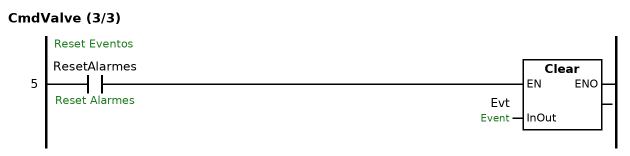
(* [picture p168: CmdValve, rungs 5-5] *)
(* Rung 5: Reset Eventos *)
IF ResetAlarmes THEN Clear(InOut := Evt); END_IF;
END_FUNCTION_BLOCK

FUNCTION_BLOCK CheckAlarmeEquip
VAR_IN_OUT
    Alm : Alarme;  (* Alarme *)
END_VAR
VAR_OUTPUT
    AlmOut : BOOL;  (* Output Alarme Agrupado *)
END_VAR
VAR_INPUT
    Enable : BOOL;
END_VAR
VAR_EXTERNAL
    ResetAlarmes : BOOL;
END_VAR
(* ladder, written here as Structured Text *)

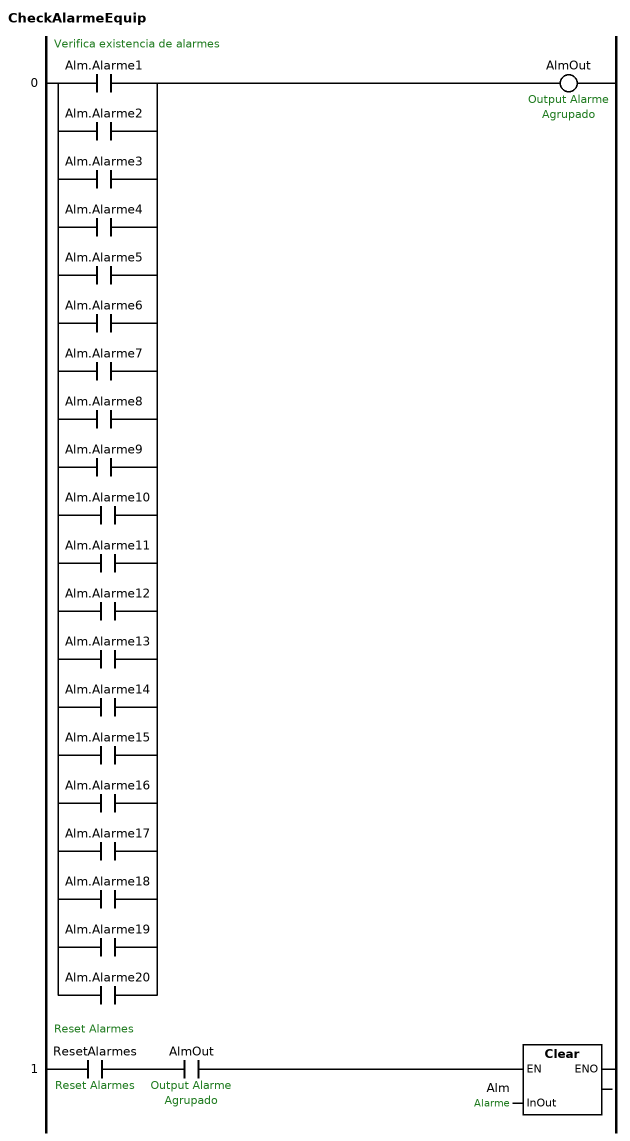
(* Rung 0: Verifica existencia de alarmes *)
AlmOut := Alm.Alarme1 OR Alm.Alarme2 OR Alm.Alarme3 OR Alm.Alarme4 OR Alm.Alarme5 OR Alm.Alarme6 OR Alm.Alarme7 OR Alm.Alarme8 OR Alm.Alarme9 OR Alm.Alarme10 OR Alm.Alarme11 OR Alm.Alarme12 OR Alm.Alarme13 OR Alm.Alarme14 OR Alm.Alarme15 OR Alm.Alarme16 OR Alm.Alarme17 OR Alm.Alarme18 OR Alm.Alarme19 OR Alm.Alarme20;
(* Rung 1: Reset Alarmes *)
IF ResetAlarmes AND AlmOut THEN Clear(InOut := Alm); END_IF;
END_FUNCTION_BLOCK

FUNCTION_BLOCK TimerPulse
VAR
    AuxTimeCalc : UINT;
END_VAR
VAR_INPUT
    Enable : BOOL;
    Pulse : BOOL;
    SetpointTime : UINT;
END_VAR
VAR
    _e1 : R_TRIG;
END_VAR
(* ladder, written here as Structured Text *)

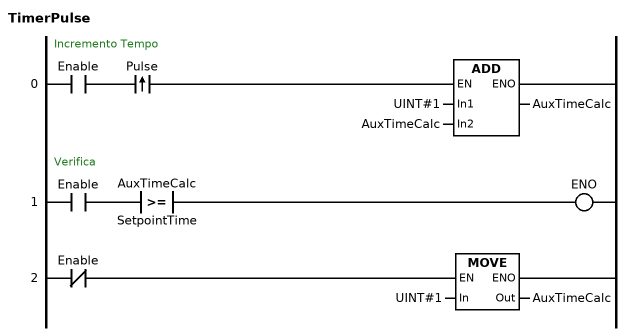
(* Rung 0: Incremento Tempo *)
_e1(CLK := Pulse);
IF Enable AND _e1.Q THEN AuxTimeCalc := UINT#1 + AuxTimeCalc; END_IF;
(* Rung 1: Verifica *)
ENO := Enable AND (AuxTimeCalc >= SetpointTime);
(* Rung 2 *)
IF NOT Enable THEN AuxTimeCalc := UINT#1; END_IF;
END_FUNCTION_BLOCK

FUNCTION_BLOCK EAN13Read
VAR
    SomaPares : UINT;
    SomaImpares : UINT;
    Resto : UINT;
    G_Step05 : BOOL;
    ResSoma : UINT;
    CodeAtCodeReader_01 : String[2];
    CodeAtCodeReader_02 : String[2];
    CodeAtCodeReader_03 : String[2];
    CodeAtCodeReader_04 : String[2];
    CodeAtCodeReader_05 : String[2];
    CodeAtCodeReader_06 : String[2];
    CodeAtCodeReader_07 : String[2];
    CodeAtCodeReader_08 : String[2];
    CodeAtCodeReader_09 : String[2];
    CodeAtCodeReader_10 : String[2];
    CodeAtCodeReader_11 : String[2];
    CodeAtCodeReader_12 : String[2];
    CodeAtCodeReader_13 : String[2];
    CodeAtCodeReader : string[128];
    TriggerTimer : TON;
    Center : UINT;
    ZeroDigit : UINT;
    CheckDigit : UINT;
    CodeValid_OK : BOOL;  (* Code Result is Valid *)
    CodeValid_NOK : BOOL;  (* Code Result is Not Valid *)
    G_Step01 : BOOL;
    G_Step02 : BOOL;
    G_Step03 : BOOL;
    G_Step04 : BOOL;
    G_Step00 : BOOL;
    G_Step06 : BOOL;
    TP_0502 : TP;
    TP_0501 : TP;
    DelayToCalc : TON;
    G_Step025 : BOOL;
    Digit : ARRAY[0..13] OF UINT;
    DigitTemp : ARRAY[0..13] OF BYTE;
    Restochk : UINT;
END_VAR
VAR_OUTPUT
    TriggerOut : BOOL;  (* Trigger para Sensor e iluminacao *)
END_VAR
VAR_INPUT
    RetentiveTimer : TIME;
    Enable : BOOL;
END_VAR
VAR_IN_OUT
    ClearData : BOOL;
END_VAR
VAR_INPUT
    Trigger : BOOL;
END_VAR
VAR_OUTPUT
    ProductRef : UINT;
    BpsId : UINT;
    ProductSeqNr : UINT;
    JulianDate : UINT;
    Year : UINT;
END_VAR
VAR_INPUT
    IFM_BarCode : ARRAY[0..449] OF BYTE;
END_VAR
VAR_OUTPUT
    EAN13 : STRING[128];
    BarCodeOK : BOOL;  (* BarCode Data OK *)
    BarCodeNOK : BOOL;  (* BarCode Data NOT OK *)
END_VAR
VAR_INPUT
    ReadOk : BOOL;
END_VAR
VAR_OUTPUT
    ET_RetentiveTimer : TIME;
END_VAR
VAR
    _e1 : R_TRIG;
    _e2 : R_TRIG;
    _p3 : BOOL;
    _p4 : BOOL;
END_VAR
(* ladder, written here as Structured Text *)

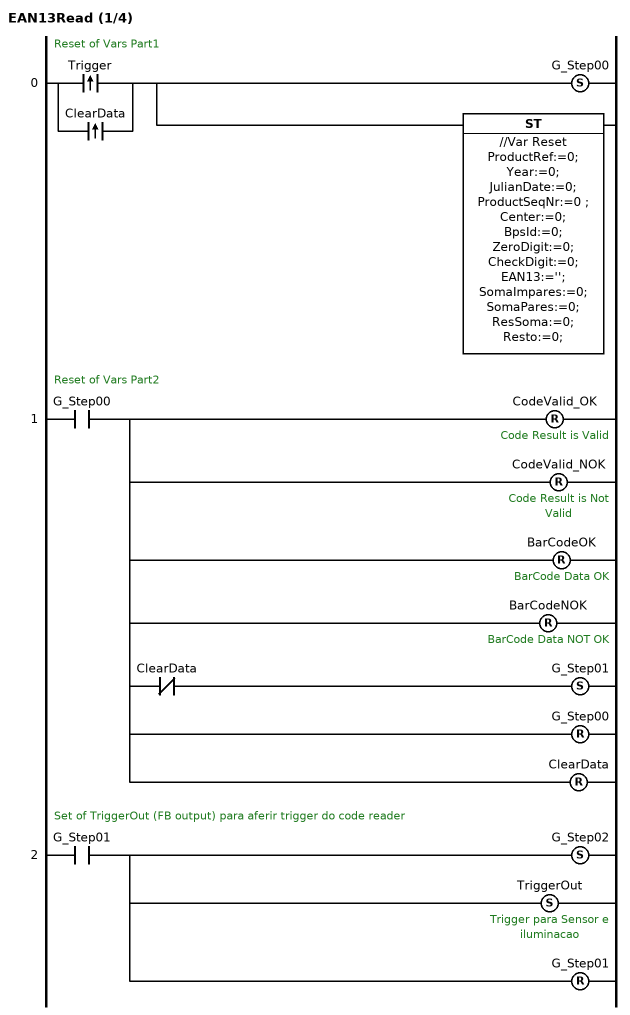
(* Rung 0: Reset of Vars Part1 *)
_e1(CLK := Trigger);
_e2(CLK := ClearData);
IF _e1.Q OR _e2.Q THEN G_Step00 := TRUE; END_IF;
IF _e1.Q OR _e2.Q THEN
    //Var Reset
    ProductRef:=0;	
    Year:=0;
    JulianDate:=0;
    ProductSeqNr:=0	;
    Center:=0;	
    BpsId:=0;	
    ZeroDigit:=0;
    CheckDigit:=0;
    EAN13:='';
    SomaImpares:=0;
    SomaPares:=0;
    ResSoma:=0;
    Resto:=0;
END_IF;
(* Rung 1: Reset of Vars Part2 *)
IF G_Step00 THEN
    CodeValid_OK := FALSE;
    CodeValid_NOK := FALSE;
    BarCodeOK := FALSE;
    BarCodeNOK := FALSE;
END_IF;
IF G_Step00 AND NOT ClearData THEN G_Step01 := TRUE; END_IF;
_p3 := G_Step00;
IF _p3 THEN
    G_Step00 := FALSE;
    ClearData := FALSE;
END_IF;
(* Rung 2: Set of TriggerOut (FB output) para aferir trigger do code reader *)
IF G_Step01 THEN
    G_Step02 := TRUE;
    TriggerOut := TRUE;
    G_Step01 := FALSE;
END_IF;

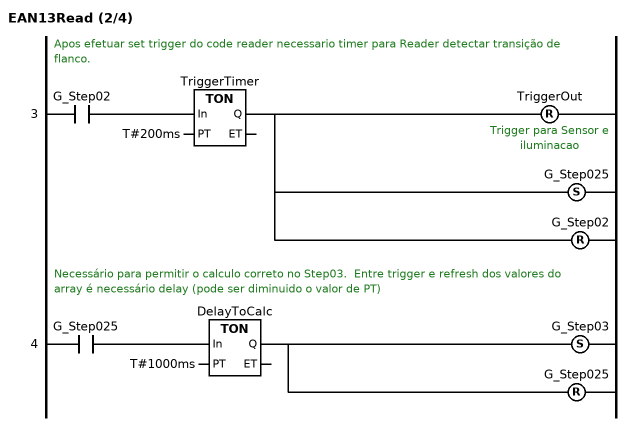
(* Rung 3: Apos efetuar set trigger do code reader necessario timer para Reader detectar transição de flanco. *)
TriggerTimer(In := G_Step02, PT := T#200ms);
IF TriggerTimer.Q THEN
    TriggerOut := FALSE;
    G_Step025 := TRUE;
    G_Step02 := FALSE;
END_IF;
(* Rung 4: Necessário para permitir o calculo correto no Step03.  Entre trigger e refresh dos valores do array é necessário delay (pode ser diminuido o valor de PT) *)
DelayToCalc(In := G_Step025, PT := T#1000ms);
IF DelayToCalc.Q THEN
    G_Step03 := TRUE;
    G_Step025 := FALSE;
END_IF;

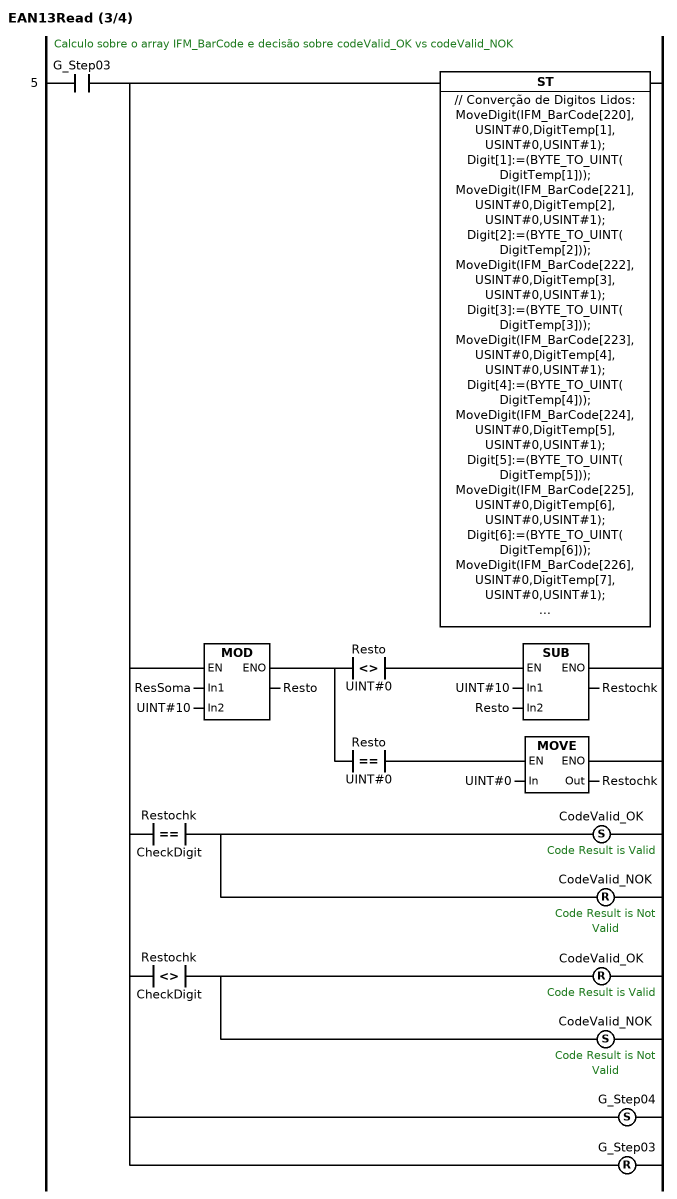
(* Rung 5: Calculo sobre o array IFM_BarCode e decisão sobre codeValid_OK vs codeValid_NOK *)
IF G_Step03 THEN
    // Converção de Digitos Lidos:
    MoveDigit(IFM_BarCode[220],USINT#0,DigitTemp[1],USINT#0,USINT#1);
    Digit[1]:=(BYTE_TO_UINT(DigitTemp[1]));
    MoveDigit(IFM_BarCode[221],USINT#0,DigitTemp[2],USINT#0,USINT#1);
    Digit[2]:=(BYTE_TO_UINT(DigitTemp[2]));
    MoveDigit(IFM_BarCode[222],USINT#0,DigitTemp[3],USINT#0,USINT#1);
    Digit[3]:=(BYTE_TO_UINT(DigitTemp[3]));
    MoveDigit(IFM_BarCode[223],USINT#0,DigitTemp[4],USINT#0,USINT#1);
    Digit[4]:=(BYTE_TO_UINT(DigitTemp[4]));
    MoveDigit(IFM_BarCode[224],USINT#0,DigitTemp[5],USINT#0,USINT#1);
    Digit[5]:=(BYTE_TO_UINT(DigitTemp[5]));
    MoveDigit(IFM_BarCode[225],USINT#0,DigitTemp[6],USINT#0,USINT#1);
    Digit[6]:=(BYTE_TO_UINT(DigitTemp[6]));
    MoveDigit(IFM_BarCode[226],USINT#0,DigitTemp[7],USINT#0,USINT#1);
    Digit[7]:=(BYTE_TO_UINT(DigitTemp[7]));
    MoveDigit(IFM_BarCode[227],USINT#0,DigitTemp[8],USINT#0,USINT#1);
    Digit[8]:=(BYTE_TO_UINT(DigitTemp[8]));
    MoveDigit(IFM_BarCode[228],USINT#0,DigitTemp[9],USINT#0,USINT#1);
    Digit[9]:=(BYTE_TO_UINT(DigitTemp[9]));
    MoveDigit(IFM_BarCode[229],USINT#0,DigitTemp[10],USINT#0,USINT#1);
    Digit[10]:=(BYTE_TO_UINT(DigitTemp[10]));
    MoveDigit(IFM_BarCode[230],USINT#0,DigitTemp[11],USINT#0,USINT#1);
    Digit[11]:=(BYTE_TO_UINT(DigitTemp[11]));
    MoveDigit(IFM_BarCode[231],USINT#0,DigitTemp[12],USINT#0,USINT#1);
    Digit[12]:=(BYTE_TO_UINT(DigitTemp[12]));
    MoveDigit(IFM_BarCode[232],USINT#0,DigitTemp[13],USINT#0,USINT#1);
    Digit[13]:=(BYTE_TO_UINT(DigitTemp[13]));
    
    
    //Checkdigit EAN13:
    SomaImpares:=3*(Digit[2]+Digit[4]+Digit[6]+Digit[8]+Digit[10]+Digit[12]);
    SomaPares:=(Digit[1]+Digit[3]+Digit[5]+Digit[7]+Digit[9]+Digit[11]);
    ResSoma:=SomaImpares+SomaPares;
    CheckDigit:=Digit[13];
END_IF;
IF G_Step03 THEN Resto := ResSoma MOD UINT#10; END_IF;
IF G_Step03 AND (Resto <> UINT#0) THEN Restochk := UINT#10 - Resto; END_IF;
IF G_Step03 AND (Resto = UINT#0) THEN Restochk := UINT#0; END_IF;
IF G_Step03 AND (Restochk = CheckDigit) THEN
    CodeValid_OK := TRUE;
    CodeValid_NOK := FALSE;
END_IF;
IF G_Step03 AND (Restochk <> CheckDigit) THEN
    CodeValid_OK := FALSE;
    CodeValid_NOK := TRUE;
END_IF;
IF G_Step03 THEN
    G_Step04 := TRUE;
    G_Step03 := FALSE;
END_IF;

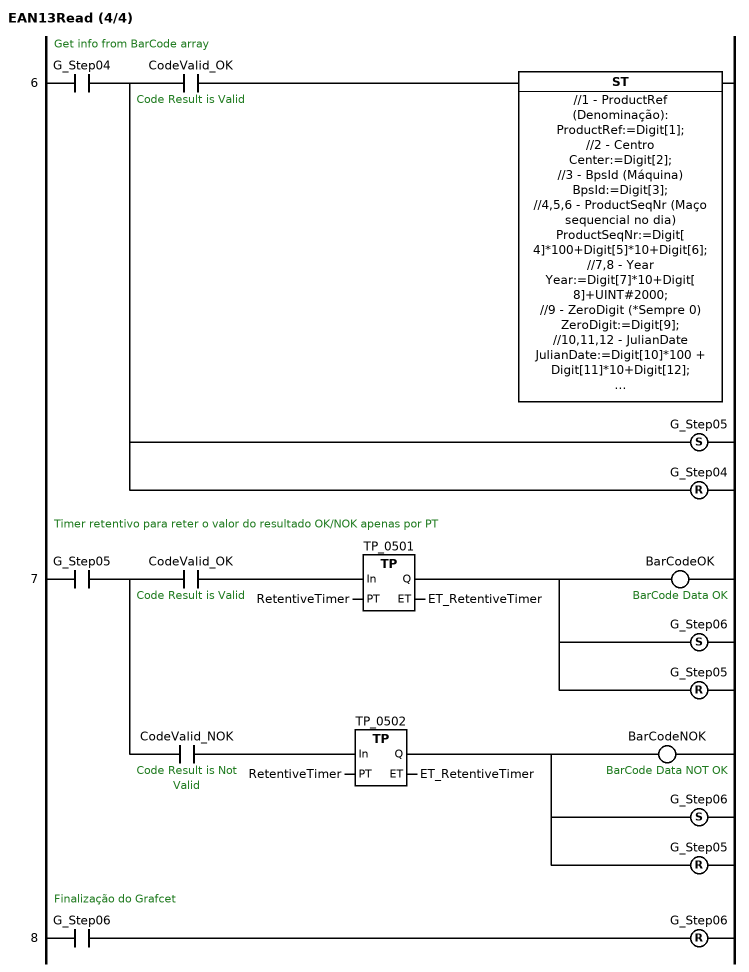
(* Rung 6: Get info from BarCode array *)
IF G_Step04 AND CodeValid_OK THEN
    //1 - ProductRef (Denominação):
    ProductRef:=Digit[1];
    //2 - Centro
    Center:=Digit[2];
    //3 - BpsId (Máquina)
    BpsId:=Digit[3];
    //4,5,6 - ProductSeqNr (Maço sequencial no dia)
    ProductSeqNr:=Digit[4]*100+Digit[5]*10+Digit[6];
    //7,8 - Year
    Year:=Digit[7]*10+Digit[8]+UINT#2000;
    //9 - ZeroDigit (*Sempre 0)
    ZeroDigit:=Digit[9];
    //10,11,12 - JulianDate
    JulianDate:=Digit[10]*100 + Digit[11]*10+Digit[12];
    
    
    //Não alterado pois é TO_INT e não TO_UINT
    //Conversão para caracter Byte a Byte (visto que hmi necessita string)
    IntAscii2Char( BYTE_TO_INT(IFM_BarCode[220]),CodeAtCodeReader_01);
    IntAscii2Char( BYTE_TO_INT(IFM_BarCode[221]),CodeAtCodeReader_02);
    IntAscii2Char( BYTE_TO_INT(IFM_BarCode[222]),CodeAtCodeReader_03);
    IntAscii2Char( BYTE_TO_INT(IFM_BarCode[223]),CodeAtCodeReader_04);
    IntAscii2Char( BYTE_TO_INT(IFM_BarCode[224]),CodeAtCodeReader_05);
    IntAscii2Char( BYTE_TO_INT(IFM_BarCode[225]),CodeAtCodeReader_06);
    IntAscii2Char( BYTE_TO_INT(IFM_BarCode[226]),CodeAtCodeReader_07);
    IntAscii2Char( BYTE_TO_INT(IFM_BarCode[227]),CodeAtCodeReader_08);
    IntAscii2Char( BYTE_TO_INT(IFM_BarCode[228]),CodeAtCodeReader_09);
    IntAscii2Char( BYTE_TO_INT(IFM_BarCode[229]),CodeAtCodeReader_10);
    IntAscii2Char( BYTE_TO_INT(IFM_BarCode[230]),CodeAtCodeReader_11);
    IntAscii2Char( BYTE_TO_INT(IFM_BarCode[231]),CodeAtCodeReader_12);
    IntAscii2Char( BYTE_TO_INT(IFM_BarCode[232]),CodeAtCodeReader_13);
    
    //String total
    CodeAtCodeReader:='';
    CodeAtCodeReader:=CONCAT(CodeAtCodeReader,CodeAtCodeReader_01);
    CodeAtCodeReader:=CONCAT(CodeAtCodeReader,CodeAtCodeReader_02);
    CodeAtCodeReader:=CONCAT(CodeAtCodeReader,CodeAtCodeReader_03);
    CodeAtCodeReader:=CONCAT(CodeAtCodeReader,CodeAtCodeReader_04);
    CodeAtCodeReader:=CONCAT(CodeAtCodeReader,CodeAtCodeReader_05);
    CodeAtCodeReader:=CONCAT(CodeAtCodeReader,CodeAtCodeReader_06);
    CodeAtCodeReader:=CONCAT(CodeAtCodeReader,CodeAtCodeReader_07);
    CodeAtCodeReader:=CONCAT(CodeAtCodeReader,CodeAtCodeReader_08);
    CodeAtCodeReader:=CONCAT(CodeAtCodeReader,CodeAtCodeReader_09);
    CodeAtCodeReader:=CONCAT(CodeAtCodeReader,CodeAtCodeReader_10);
    CodeAtCodeReader:=CONCAT(CodeAtCodeReader,CodeAtCodeReader_11);
    CodeAtCodeReader:=CONCAT(CodeAtCodeReader,CodeAtCodeReader_12);
    CodeAtCodeReader:=CONCAT(CodeAtCodeReader,CodeAtCodeReader_13);
    
    //EAN 13 ja convertido para String
    EAN13:=CodeAtCodeReader;
END_IF;
IF G_Step04 THEN
    G_Step05 := TRUE;
    G_Step04 := FALSE;
END_IF;
(* Rung 7: Timer retentivo para reter o valor do resultado OK/NOK apenas por PT *)
TP_0501(In := G_Step05 AND CodeValid_OK, PT := RetentiveTimer, ET => ET_RetentiveTimer);
BarCodeOK := TP_0501.Q;
IF TP_0501.Q THEN G_Step06 := TRUE; END_IF;
_p4 := G_Step05;
IF TP_0501.Q THEN G_Step05 := FALSE; END_IF;
TP_0502(In := _p4 AND CodeValid_NOK, PT := RetentiveTimer, ET => ET_RetentiveTimer);
BarCodeNOK := TP_0502.Q;
IF TP_0502.Q THEN
    G_Step06 := TRUE;
    G_Step05 := FALSE;
END_IF;
(* Rung 8: Finalização do Grafcet *)
IF G_Step06 THEN G_Step06 := FALSE; END_IF;
END_FUNCTION_BLOCK

FUNCTION_BLOCK CheckBarCode
VAR_IN_OUT
    Alm : Alarme;  (* Alarme *)
END_VAR
VAR_OUTPUT
    AlmOut : BOOL;  (* Output Alarme Agrupado *)
END_VAR
VAR_INPUT
    Enable : BOOL;
    Reset : BOOL;
END_VAR
(* ladder, written here as Structured Text *)

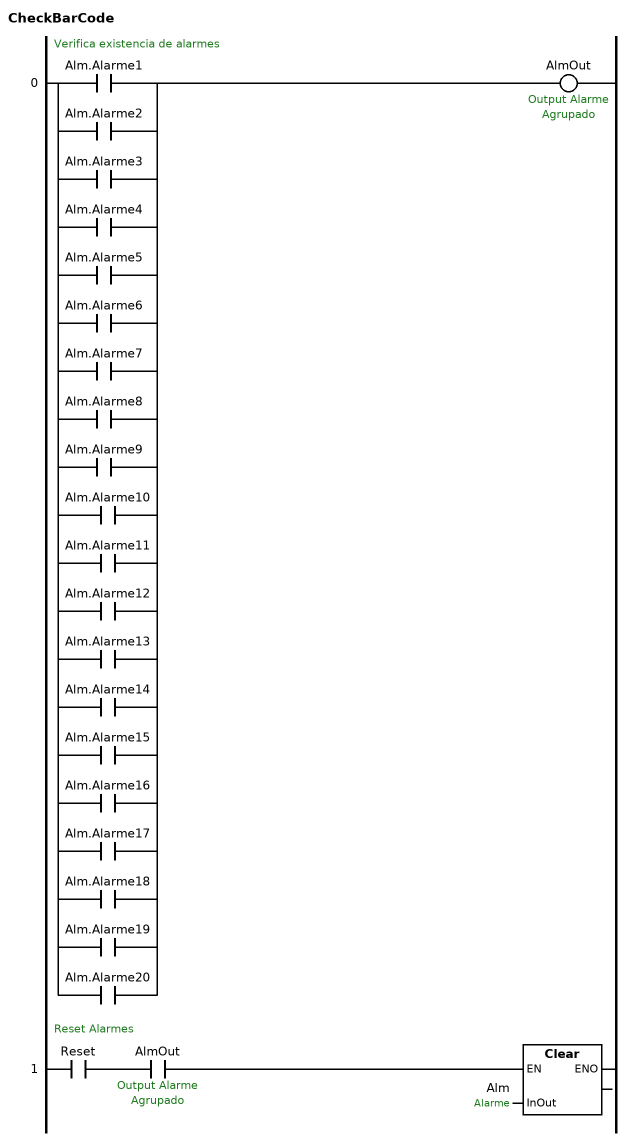
(* Rung 0: Verifica existencia de alarmes *)
AlmOut := Alm.Alarme1 OR Alm.Alarme2 OR Alm.Alarme3 OR Alm.Alarme4 OR Alm.Alarme5 OR Alm.Alarme6 OR Alm.Alarme7 OR Alm.Alarme8 OR Alm.Alarme9 OR Alm.Alarme10 OR Alm.Alarme11 OR Alm.Alarme12 OR Alm.Alarme13 OR Alm.Alarme14 OR Alm.Alarme15 OR Alm.Alarme16 OR Alm.Alarme17 OR Alm.Alarme18 OR Alm.Alarme19 OR Alm.Alarme20;
(* Rung 1: Reset Alarmes *)
IF Reset AND AlmOut THEN Clear(InOut := Alm); END_IF;
END_FUNCTION_BLOCK

FUNCTION_BLOCK CmdICM
VAR_INPUT
    Enable : BOOL;
    I_Interroll : In_EIPMulticontrol;
END_VAR
VAR_OUTPUT
    Q_Interroll : Out_EIPMulticontrol;
END_VAR
VAR_INPUT
    NotExternAlarm : BOOL;
END_VAR
VAR_OUTPUT
    Alarm_01 : AlarmeGeralEquipamento;
    Alarm_02 : AlarmeGeralEquipamento;
    Alarm_03 : AlarmeGeralEquipamento;
    Alarm_04 : AlarmeGeralEquipamento;
    Sensor_01 : BOOL;
    IO_01 : BOOL;
    Sensor_02 : BOOL;
    IO_02 : BOOL;
    Sensor_03 : BOOL;
    IO_03 : BOOL;
    Sensor_04 : BOOL;
    IO_04 : BOOL;
END_VAR
VAR_INPUT
    DataMotor_01 : DataMotor;
    DataMotor_02 : DataMotor;
    DataMotor_03 : DataMotor;
    DataMotor_04 : DataMotor;
END_VAR
VAR_EXTERNAL
    ResetAlarmes : BOOL;
END_VAR
(* ladder, written here as Structured Text *)

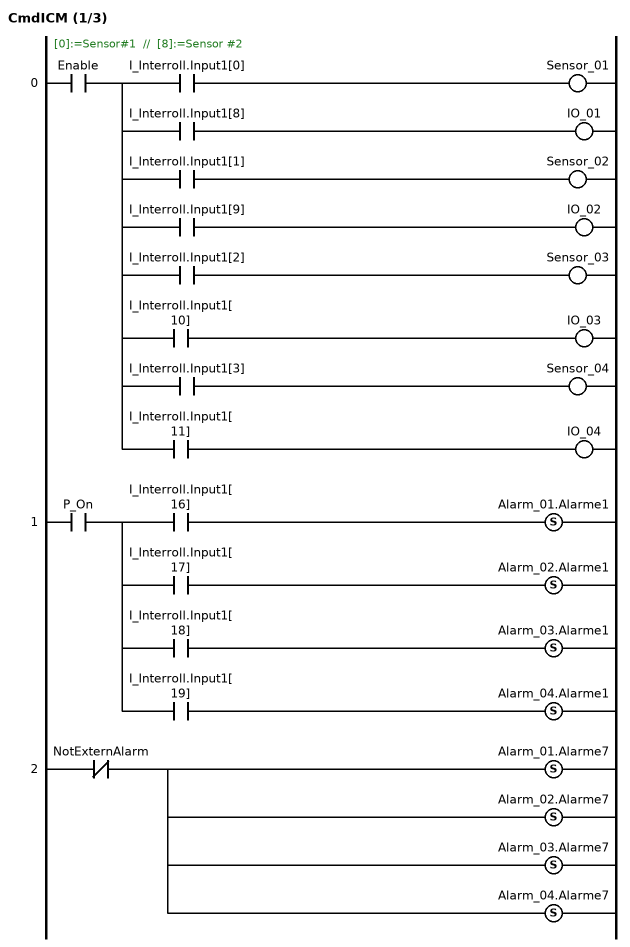
(* Rung 0: [0]:=Sensor#1  //  [8]:=Sensor #2 *)
Sensor_01 := Enable AND I_Interroll.Input1[0];
IO_01 := Enable AND I_Interroll.Input1[8];
Sensor_02 := Enable AND I_Interroll.Input1[1];
IO_02 := Enable AND I_Interroll.Input1[9];
Sensor_03 := Enable AND I_Interroll.Input1[2];
IO_03 := Enable AND I_Interroll.Input1[10];
Sensor_04 := Enable AND I_Interroll.Input1[3];
IO_04 := Enable AND I_Interroll.Input1[11];
(* Rung 1 *)
IF P_On AND I_Interroll.Input1[16] THEN Alarm_01.Alarme1 := TRUE; END_IF;
IF P_On AND I_Interroll.Input1[17] THEN Alarm_02.Alarme1 := TRUE; END_IF;
IF P_On AND I_Interroll.Input1[18] THEN Alarm_03.Alarme1 := TRUE; END_IF;
IF P_On AND I_Interroll.Input1[19] THEN Alarm_04.Alarme1 := TRUE; END_IF;
(* Rung 2 *)
IF NOT NotExternAlarm THEN
    Alarm_01.Alarme7 := TRUE;
    Alarm_02.Alarme7 := TRUE;
    Alarm_03.Alarme7 := TRUE;
    Alarm_04.Alarme7 := TRUE;
END_IF;

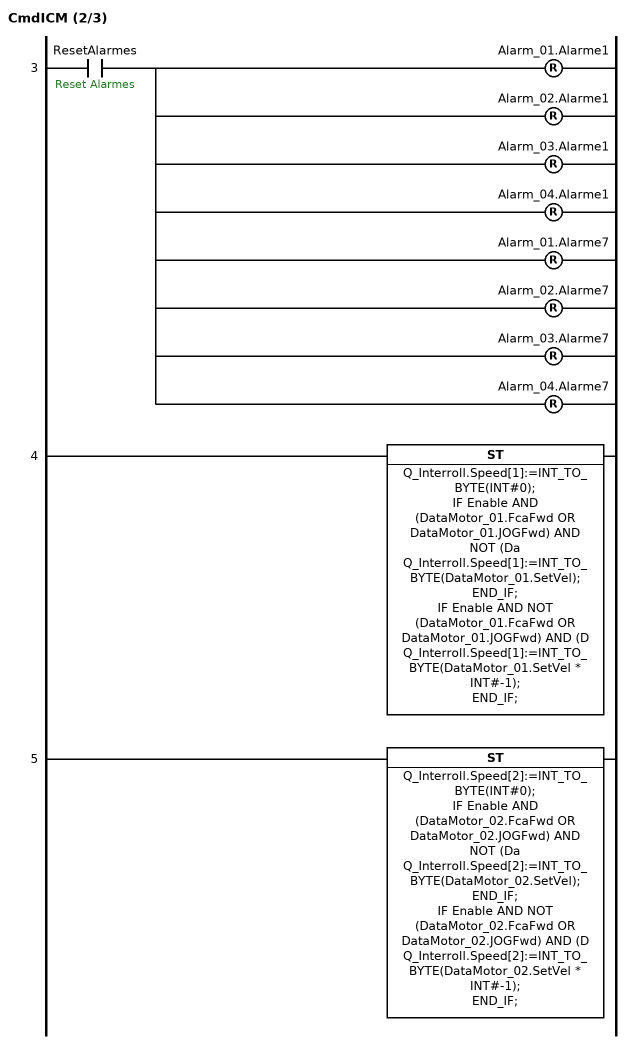
(* Rung 3 *)
IF ResetAlarmes THEN
    Alarm_01.Alarme1 := FALSE;
    Alarm_02.Alarme1 := FALSE;
    Alarm_03.Alarme1 := FALSE;
    Alarm_04.Alarme1 := FALSE;
    Alarm_01.Alarme7 := FALSE;
    Alarm_02.Alarme7 := FALSE;
    Alarm_03.Alarme7 := FALSE;
    Alarm_04.Alarme7 := FALSE;
END_IF;
(* Rung 4 *)
Q_Interroll.Speed[1]:=INT_TO_BYTE(INT#0);
IF Enable AND (DataMotor_01.FcaFwd OR DataMotor_01.JOGFwd) AND NOT (DataMotor_01.FcaRev OR DataMotor_01.JOGRev) THEN
	Q_Interroll.Speed[1]:=INT_TO_BYTE(DataMotor_01.SetVel);
END_IF;
IF Enable AND NOT  (DataMotor_01.FcaFwd OR DataMotor_01.JOGFwd) AND (DataMotor_01.FcaRev OR DataMotor_01.JOGRev) THEN
	Q_Interroll.Speed[1]:=INT_TO_BYTE(DataMotor_01.SetVel * INT#-1);
END_IF;
(* Rung 5 *)
Q_Interroll.Speed[2]:=INT_TO_BYTE(INT#0);
IF Enable AND (DataMotor_02.FcaFwd OR DataMotor_02.JOGFwd) AND NOT (DataMotor_02.FcaRev OR DataMotor_02.JOGRev) THEN
	Q_Interroll.Speed[2]:=INT_TO_BYTE(DataMotor_02.SetVel);
END_IF;
IF Enable AND NOT  (DataMotor_02.FcaFwd OR DataMotor_02.JOGFwd) AND (DataMotor_02.FcaRev OR DataMotor_02.JOGRev) THEN
	Q_Interroll.Speed[2]:=INT_TO_BYTE(DataMotor_02.SetVel * INT#-1);
END_IF;

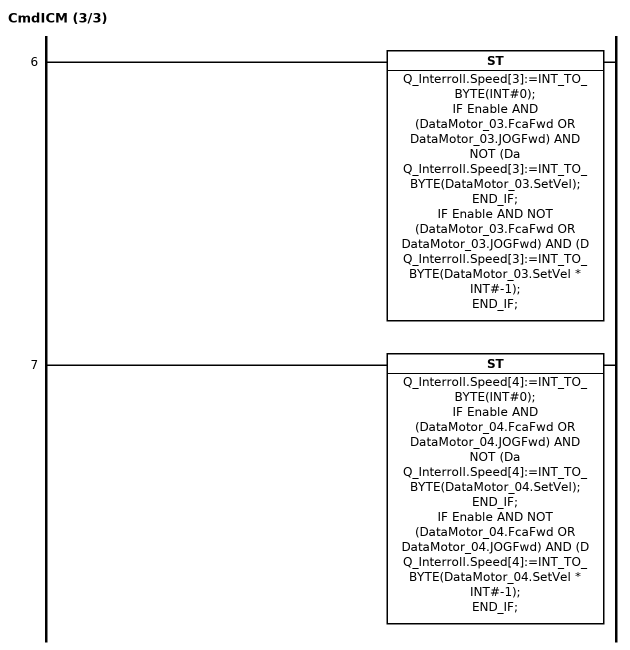
(* Rung 6 *)
Q_Interroll.Speed[3]:=INT_TO_BYTE(INT#0);
IF Enable AND (DataMotor_03.FcaFwd OR DataMotor_03.JOGFwd) AND NOT (DataMotor_03.FcaRev OR DataMotor_03.JOGRev) THEN
	Q_Interroll.Speed[3]:=INT_TO_BYTE(DataMotor_03.SetVel);
END_IF;
IF Enable AND NOT  (DataMotor_03.FcaFwd OR DataMotor_03.JOGFwd) AND (DataMotor_03.FcaRev OR DataMotor_03.JOGRev) THEN
	Q_Interroll.Speed[3]:=INT_TO_BYTE(DataMotor_03.SetVel * INT#-1);
END_IF;
(* Rung 7 *)
Q_Interroll.Speed[4]:=INT_TO_BYTE(INT#0);
IF Enable AND (DataMotor_04.FcaFwd OR DataMotor_04.JOGFwd) AND NOT (DataMotor_04.FcaRev OR DataMotor_04.JOGRev) THEN
	Q_Interroll.Speed[4]:=INT_TO_BYTE(DataMotor_04.SetVel);
END_IF;
IF Enable AND NOT  (DataMotor_04.FcaFwd OR DataMotor_04.JOGFwd) AND (DataMotor_04.FcaRev OR DataMotor_04.JOGRev) THEN
	Q_Interroll.Speed[4]:=INT_TO_BYTE(DataMotor_04.SetVel * INT#-1);
END_IF;
END_FUNCTION_BLOCK